// TIA Portal V16 export
// export: Created 2021-07-12T14:47:08.2591518Z, ExportSetting WithDefaults, DisplayName Totally Integrated Automation Portal, DisplayVersion V16, DisplayName TIA Portal Version Control Interface, DisplayVersion V16, DisplayName TIA Portal Openness, DisplayVersion V16, DisplayName STEP 7 Professional, DisplayVersion V16, DisplayName STEP 7 Safety, DisplayVersion V16, DisplayName WinCC Professional, DisplayVersion V16
FUNCTION_BLOCK "SimaHydTO_AxisBasics_SyncAxis"   // FB33193, FBD
TITLE = SimaHydTO_AxisBasics_SyncAxis
{ S7_Optimized_Access := 'TRUE' }
FAMILY : SimaHydTO/LAxisBasics
VERSION : 1.0
// Function block information: See Function block network 1
// stored: AutoNumber true, IsIECCheckEnabled false, IsRetainMemResEnabled false, MemoryReserve 100, SetENOAutomatically false, UDAEnableTagReadback false
   VAR_INPUT
      axis : TO_SynchronousAxis;   // Technology object (axis)
      powerEnable : Bool;   // MC_Power: 0: The technology object is disabled / 1: The technology object is enabled
      powerStartMode : DInt := 1;   // 0: Enable axis not position-controlled / 1: Enable axis position-controlled
      powerStopMode : Int := 0;   // 0: Emergency stop / 1: Immediate stop / 2: Stop with maximum dynamic values
      resetExecute : Bool;   // MC_Reset: Start job with a positive edge
      resetRestart : Bool := false;   // 0: Acknowledgment of queued technology alarms / 1: Reinitialization of the technology object and acknowledgment of pending technology alarms
      homeExecute : Bool;   // MC_Home: Start job with a positive edge
      homePosition : LReal;   // The specified value is used according to the selected "Mode".
      homeMode : Int;   // 0: Direct homing (absolute) / 1: Direct homing (relative) / 2: Passive homing / 3: Active homing / 4: Reserved / 5: Active homing (<TO>.Homing.HomePosition) / 6: Absolute encoder adjustment (relative) / 7: Absolute encoder adjustment (absolute) / 8: Passive homing / 9: Abort passive homing / 10: Passive homing (<TO>.Homing.HomePosition)
      jogForward : Bool;   // MC_MoveJog: As long as the parameter is TRUE, the axis moves in the positive direction
      jogBackward : Bool;   // MC_MoveJog: As long as the parameter is TRUE, the axis moves in the negative direction
      jogVelocity : LReal := 100.0;   // Velocity setpoint / speed setpoint for the motion
      jogAcceleration : LReal := -1.0;   // Acceleration of jog movement
      jogDeceleration : LReal := -1.0;   // Deceleration of jog movement
      jogJerk : LReal := -1.0;   // Jerk of jog movement
      jogPositionControlled : Bool := true;   // 0: Non position-controlled operation / 1: Position-controlled mode - The parameter applies as long as the MC_MoveJog command is executed. After this, the setting of MC_Power applies again.
   END_VAR
   VAR_OUTPUT
      powerStatus { ExternalWritable := 'False'} : Bool;   // MC_Power: 0: Technology object disabled / 1: Technology object enabled
      powerBusy { ExternalWritable := 'False'} : Bool;   // MC_Power: Job is running
      resetDone { ExternalWritable := 'False'} : Bool;   // MC_Reset: Error has been acknowledged or Restart has been executed.
      resetBusy { ExternalWritable := 'False'} : Bool;   // MC_Reset: Job is running
      homeDone { ExternalWritable := 'False'} : Bool;   // MC_Home: Job is completed
      homeBusy { ExternalWritable := 'False'} : Bool;   // MC_Home: Job is running
      jogInVelocity { ExternalWritable := 'False'} : Bool;   // MC_MoveJog: The velocity setpoint / speed setpoint was reached and will be maintained
      jogBusy { ExternalWritable := 'False'} : Bool;   // MC_MoveJog: Job is running
      commandAborted { ExternalWritable := 'False'} : Bool;   // The job was aborted by another job during execution (see also StatusID)
      error { ExternalWritable := 'False'} : Bool;   // An error occurred during execution of the job. The job is rejected. The cause of the error can be found in the "ErrorID" parameter.
      errorID { ExternalWritable := 'False'} : Word;   // ErrorID of motion control instruction (see also StatusID)
      statusID { ExternalWritable := 'False'} : Int;   // Additional specification of affected Motion control instruction of CommandAborted or Error: 0: No instruction / 1: MC_Power / 2: MC_Reset / 3: MC_Home / 4: MC_MoveJog
   END_VAR
   VAR
      instMcPower { ExternalAccessible := 'False'; ExternalVisible := 'False'; ExternalWritable := 'False'; S7_SetPoint := 'True'} : MC_POWER;   // PLCopen functions of basic motion control
      instMcReset { ExternalAccessible := 'False'; ExternalVisible := 'False'; ExternalWritable := 'False'; S7_SetPoint := 'True'} : MC_RESET;
      instMcHome { ExternalAccessible := 'False'; ExternalVisible := 'False'; ExternalWritable := 'False'; S7_SetPoint := 'True'} : MC_HOME;
      instMcMoveJog { ExternalAccessible := 'False'; ExternalVisible := 'False'; ExternalWritable := 'False'; S7_SetPoint := 'True'} : MC_MOVEJOG;
      statCommandAborted { ExternalAccessible := 'False'; ExternalVisible := 'False'; ExternalWritable := 'False'} : Array[#ARRAY_BEGIN..#ARRAY_END] of Bool;   // Arrays to save error information of PLCopen functions
      statError { ExternalAccessible := 'False'; ExternalVisible := 'False'; ExternalWritable := 'False'} : Array[#ARRAY_BEGIN..#ARRAY_END] of Bool;
      statErrorID { ExternalAccessible := 'False'; ExternalVisible := 'False'; ExternalWritable := 'False'} : Array[#ARRAY_BEGIN..#ARRAY_END] of Word;
   END_VAR
   VAR_TEMP
      tempDwordCommandAborted : DWord;   // Variables to check error informations of PLCopen functions
      tempDwordError : DWord;
      tempCount : Int;   // Counter of FOR counting loop
   END_VAR
   VAR CONSTANT
      ARRAY_BEGIN : Int := 1;   // Start-Index of array (Maximum 32 Array elements!)
      ARRAY_END : Int := 32;   // End-Index of array (Maximum 32 Array elements!)
      ERROR_DEFAULT : Bool := false;   // Default values of output signals
      ERRORID_DEFAULT : Word := 16#0;
      STATUSID_DEFAULT : Int := 0;
   END_VAR
BEGIN

REGION Network 1 (SCL): Axis Basics - Header
   //=============================================================================
   //SIEMENS AG
   //(c)Copyright 2016 All Rights Reserved
   //-----------------------------------------------------------------------------
   //Library:       AxisBasics
   //Tested with:   S7-1500 V2.5
   //Engineering:   TIA Portal V15
   //Restrictions:  Motion Control Library V4.0
   //Requirements:  S7-1500(T)
   //Functionality: Basic axis control of TO_SynchronousAxis
   //-----------------------------------------------------------------------------
   //Change log table:
   //Version  Date       Expert in charge Changes applied
   //01.00.00 04.10.2018 ArSc             First released version
   //=============================================================================
END_REGION

REGION Network 2: Axis Basics - MC_Power
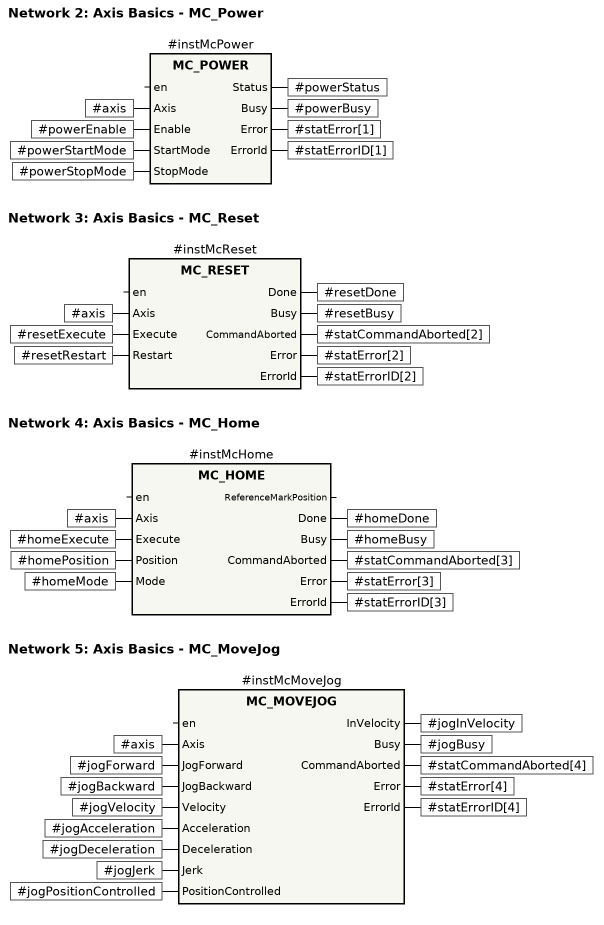
   #instMcPower(Axis := #axis,   // MC_POWER
                Enable := #powerEnable,
                StartMode := #powerStartMode,
                StopMode := #powerStopMode,
                Status => #powerStatus,
                Busy => #powerBusy,
                Error => #statError[1],
                ErrorId => #statErrorID[1]);
END_REGION

REGION Network 3: Axis Basics - MC_Reset
   #instMcReset(Axis := #axis,   // MC_RESET
                Execute := #resetExecute,
                Restart := #resetRestart,
                Done => #resetDone,
                Busy => #resetBusy,
                CommandAborted => #statCommandAborted[2],
                Error => #statError[2],
                ErrorId => #statErrorID[2]);
END_REGION

REGION Network 4: Axis Basics - MC_Home
   #instMcHome(Axis := #axis,   // MC_HOME
               Execute := #homeExecute,
               Position := #homePosition,
               Mode := #homeMode,
               Done => #homeDone,
               Busy => #homeBusy,
               CommandAborted => #statCommandAborted[3],
               Error => #statError[3],
               ErrorId => #statErrorID[3]);
END_REGION

REGION Network 5: Axis Basics - MC_MoveJog
   #instMcMoveJog(Axis := #axis,   // MC_MOVEJOG
                  JogForward := #jogForward,
                  JogBackward := #jogBackward,
                  Velocity := #jogVelocity,
                  Acceleration := #jogAcceleration,
                  Deceleration := #jogDeceleration,
                  Jerk := #jogJerk,
                  PositionControlled := #jogPositionControlled,
                  InVelocity => #jogInVelocity,
                  Busy => #jogBusy,
                  CommandAborted => #statCommandAborted[4],
                  Error => #statError[4],
                  ErrorId => #statErrorID[4]);
END_REGION

REGION Network 6 (SCL): Axis Basics - Generate output signals and error detection
   //General output signals

   //Reset output signals
   #commandAborted := False;
   #error := False;
   #errorID := #ERRORID_DEFAULT;
   #statusID := #STATUSID_DEFAULT;

   //Transfer ARRAY to DWORD
   GATHER(IN:=#statCommandAborted,
          OUT=>#tempDwordCommandAborted);
   GATHER(IN:=#statError,
          OUT=>#tempDwordError);

   //Check for errors or command aborts
   IF (#tempDwordError > DWORD#0)
   THEN
     //Select error information
     FOR #tempCount := #ARRAY_BEGIN TO #ARRAY_END
     DO
       IF (#statError[#tempCount] = True)
       THEN
         #error := True;
         #errorID := #statErrorID[#tempCount];
         #statusID := #tempCount;
         EXIT;
       END_IF;
     END_FOR;
   ELSIF (#tempDwordCommandAborted > DWORD#0)
   THEN
     //Select command aborted information
     FOR #tempCount := #ARRAY_BEGIN TO #ARRAY_END
     DO
       IF (#statCommandAborted[#tempCount] = True)
       THEN
         #commandAborted := True;
         #errorID := #statErrorID[#tempCount];
         #statusID := #tempCount;
         EXIT;
       END_IF;
     END_FOR;
   END_IF;
END_REGION
END_FUNCTION_BLOCK
